PROGRAM MAIN
VAR
END_VAR

END_PROGRAM

(* stored: Version 1.1.0.1, ProductVersion 3.1.4024.15
   POU MAIN: Id {bc9c3e96-a690-4690-b444-ea9323d20ce0}, SpecialFunc None *)
